// TwinCAT 3 PLC project MAS418PLC
// ProgramVersion: 3.1.4024.0
// libraries:
//   Tc2_Standard, * (Beckhoff Automation GmbH)
//   Tc2_System, * (Beckhoff Automation GmbH)
//   Tc3_Module, * (Beckhoff Automation GmbH)
//   VisuDialogs, * (System)
// project tree:
//   / GlobalTextList.TcGTLO, PlcTask.TcTTO, Visualization Manager.TcVMO (not stored)
//   POUs/ MAIN.TcPOU
//   VISUs/ Visualization.TcVIS

CONFIGURATION MAS418PLC
    RESOURCE PLC ON TwinCAT3
        TASK PlcTask(INTERVAL := T#10ms, PRIORITY := 20);
        PROGRAM MAIN WITH PlcTask : MAIN;
    END_RESOURCE
END_CONFIGURATION

// ---- POUs/MAIN.TcPOU
PROGRAM MAIN
VAR
	bEnable : BOOL;
	bStart : BOOL;
	nInt : INT := -32768;
	nUint : UINT := 65535;
	fReal : REAL := 255.255;
	sPowerstatus : STRING := 'Power Off';
	
    nFloatConversion : INT;
	fFloatConversion : LREAL;
	nHeltall : INT:= 100;
	fKomma : LREAL := 100.5;
	
END_VAR

bEnable := bStart;

nFloatConversion := nHeltall + LREAL_TO_INT(fKomma);

END_PROGRAM

// ---- GlobalTextList.TcGTLO
TEXTLIST GlobalTextList
  233 = '%f'
  938 = '%i'
  985 = '%s'
  332 = 'BOOL'
  602 = 'BOOL%i'
  605 = 'DataTypeTesting'
  560 = 'INT'
  238 = 'POWER ON'
  702 = 'REAL'
  240 = 'STRING'
  743 = 'UINT'
END_TEXTLIST

// ---- VISUs/Visualization.TcVIS
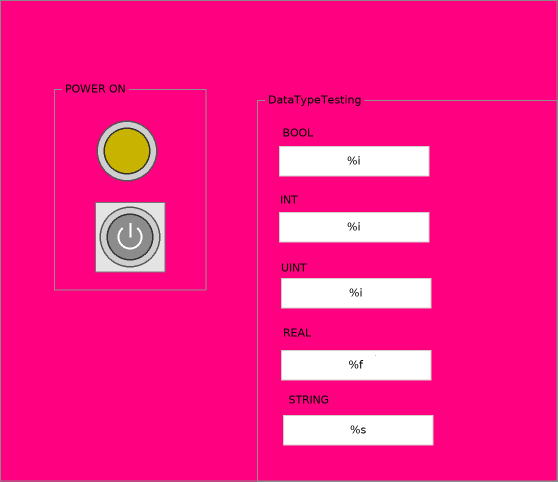
VISUALIZATION Visualization  // 558x482
    GroupBox (54,81 152x209), "POWER ON"
        Lamp1 (38,35 70x70), variable: MAIN.bEnable, style: Lamp-Lamp1-Yellow
        PowerSwitch (41,121 70x70), variable: MAIN.bStart, behaviour: TOGGLE, style: Switch-PowerSwitch-Gray
    GroupBox (257,92 301x390), "DataTypeTesting"
        Textfield (22,120 150x30), "%i", text variable: MAIN.nInt
        Textfield (22,54 150x30), "%i", text variable: MAIN.bEnable
        Textfield (24,186 150x30), "%i", text variable: MAIN.nUint
        Textfield (24,258 150x30), "%f", text variable: MAIN.fReal
            OnMouseDown: write the text variable via Edit
        Textfield (26,323 150x30), "%s", text variable: MAIN.sPowerstatus
            OnMouseDown: write the text variable via Default
            OnMouseDown: write the text variable via Default
    Label (223,118 150x30), "BOOL"
    Label (214,185 150x30), "INT"
    Label (219,253 150x30), "UINT"
    Label (222,318 150x30), "REAL"
    Label (234,385 150x30), "STRING"
    Polygon (375,355) (375,355)
END_VISUALIZATION
